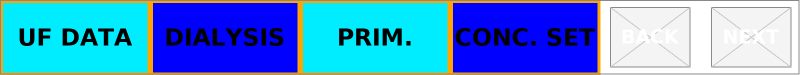
VISUALIZATION RinseMode_Footer  // 800x75
    Textfield (0,0 150x75), "UF DATA"
    Textfield (150,0 150x75), "DIALYSIS"
    Textfield (300,0 150x75), "PRIM."
    Textfield (450,0 150x75), "CONC. SET"
    Image (610,7 80x60), "BACK", image: VisuSymbols.Symbols.ArrowBoldLeft
    Image (711,7 80x60), "NEXT", image: VisuSymbols.Symbols.ArrowBoldRight
END_VISUALIZATION

(* stored: Version 1.1.0.1, ProductVersion 3.1.4024.12
   Visu RinseMode_Footer: Id {a6c3e152-2ea3-4716-a6c3-4c1f72650eac} *)
